{attribute 'hide_all_locals'}
FUNCTION_BLOCK PUBLIC FB_Utility
VAR
    CpuCounter : GETCPUCOUNTER;
END_VAR

METHOD PUBLIC GetCpuCounterAsULINT : ULINT
VAR
    TempResult : ULINT;
END_VAR
CpuCounter();
TempResult := GetCpuCounter.cpuCntHiDW;
TempResult := SHL(TempResult,32);
GetCpuCounterAsULINT := TempResult + GetCpuCounter.cpuCntLoDW;
END_METHOD

END_FUNCTION_BLOCK

(* stored: Version 1.1.0.1, ProductVersion 3.1.4022.18
   POU FB_Utility: Id {eb7474a6-4c38-44a6-a596-17f52c47b8c1}, SpecialFunc None
   Method GetCpuCounterAsULINT: Id {422b728e-cf37-4fcb-b889-112b7adf5522} *)
